(* PLC project Tc2_Utilities.FB_AddRouteEntryEx Demo, tc3-libraries-kb TwinCAT 3.1 *)
(* stored: creationDateTime 2026-05-10T20:00:00, modificationDateTime 2026-05-10T20:00:00 *)

PROGRAM P_Demo_FB_AddRouteEntryEx
  VAR
    fbFB_AddRouteEntryEx : FB_AddRouteEntryEx;  (* Tc2_Utilities.FB_AddRouteEntryEx 实例 *)
    arg_sNetID : T_AmsNetID;  (* VAR_INPUT sNetID *)
    arg_stRoute : ST_AmsRouteEntry;  (* VAR_INPUT stRoute *)
    arg_bExecute : BOOL;  (* VAR_INPUT bExecute *)
    arg_tTimeout : TIME;  (* VAR_INPUT tTimeout *)
    out_bBusy : BOOL;  (* VAR_OUTPUT bBusy *)
    out_bError : BOOL;  (* VAR_OUTPUT bError *)
    out_nErrId : UDINT;  (* VAR_OUTPUT nErrId *)
  END_VAR

            // ============================================================
// Tc2_Utilities.FB_AddRouteEntryEx 演示程序（FB 实例）
// ============================================================
// 验证步骤：
//   1. 引用 Tc2_Utilities（及依赖类型所在库 Tc2_System 等）
//   2. 编译 + 登录
//   3. 按 doc.md 给 arg_* 赋值
//   4. 在线监视 out_* / io_* 输出
// ============================================================

fbFB_AddRouteEntryEx(
    sNetID := arg_sNetID,
    stRoute := arg_stRoute,
    bExecute := arg_bExecute,
    tTimeout := arg_tTimeout,
    bBusy => out_bBusy,
    bError => out_bError,
    nErrId => out_nErrId
);

          
END_PROGRAM
